// TIA Portal V19 export
TYPE "MES_Msg_Receive_Topic3xx_Err"
// stored: Access Published
   STRUCT
      Recive_MSG300 { ExternalAccessible := 'False'; ExternalVisible := 'False'; ExternalWritable := 'False'} : "MES_Err_&_Msg";
      Recive_MSG301 { ExternalAccessible := 'False'; ExternalVisible := 'False'; ExternalWritable := 'False'} : "MES_Err_&_Msg";
   END_STRUCT;
END_TYPE
